FUNCTION_BLOCK InjectorMotorController
  (* Standard: 61499-2 *)
  (* Version 0.1, 2016-00-28, hpea485, UOA *)
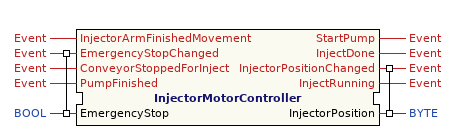
  EVENT_INPUT
    InjectorArmFinishedMovement;
    EmergencyStopChanged WITH EmergencyStop;
    ConveyorStoppedForInject;
    PumpFinished;
  END_EVENT
  EVENT_OUTPUT
    StartPump;
    InjectDone;
    InjectorPositionChanged WITH InjectorPosition;
    InjectRunning;
  END_EVENT
  VAR_INPUT
    EmergencyStop : BOOL;
  END_VAR
  VAR_OUTPUT
    InjectorPosition : BYTE;
  END_VAR
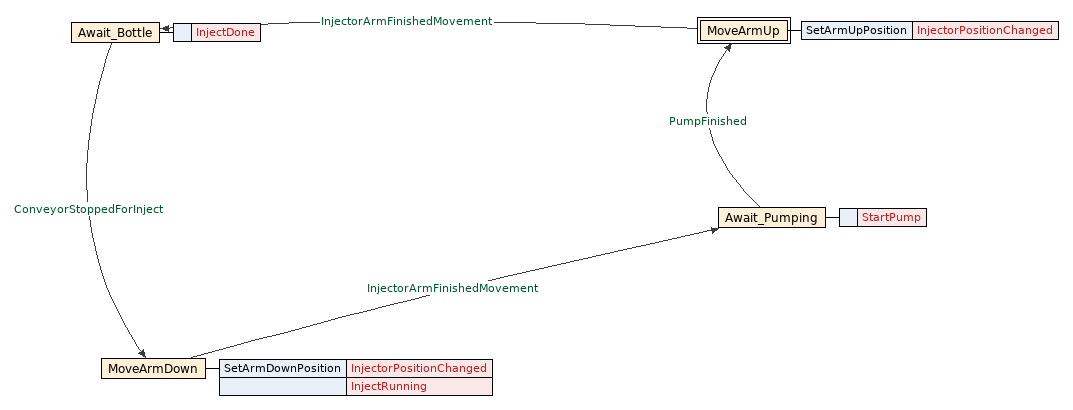
  EC_STATES
    MoveArmUp : SetArmUpPosition -> InjectorPositionChanged;
    Await_Bottle : -> InjectDone;
    MoveArmDown : SetArmDownPosition -> InjectorPositionChanged, -> InjectRunning;
    Await_Pumping : -> StartPump;
  END_STATES
  EC_TRANSITIONS
    Await_Bottle TO MoveArmDown := ConveyorStoppedForInject;
    MoveArmDown TO Await_Pumping := InjectorArmFinishedMovement;
    Await_Pumping TO MoveArmUp := PumpFinished;
    MoveArmUp TO Await_Bottle := InjectorArmFinishedMovement;
  END_TRANSITIONS
  ALGORITHM SetArmDownPosition IN C:
me->InjectorPosition = 255;
//printf("Injector: Set Injector Arm to Down position\n");
  END_ALGORITHM
  ALGORITHM SetArmUpPosition IN C:
printf("Injector: Set injector arm to up position\n");
me->InjectorPosition = 0;
  END_ALGORITHM
  ALGORITHM Algorithm1 IN C:
printf("lalalala\n");
  END_ALGORITHM
END_FUNCTION_BLOCK
